PROGRAM MAIN
VAR
	bCoinEnter 	: BOOL;
	bManual		: BOOL;
	bAuto		: BOOL;
	bLedPower	: BOOL;

	bPlainWater	: BOOL:=TRUE;
	bLedW		: BOOL;
	
	bShampoo	: BOOL:=TRUE;
	bLedS		: BOOL;

    bWax		: BOOL:=TRUE;
	bLedWx		: BOOL;
	
	tRunningTimeM	: TIME:=T#9S;
	tTimer 		: TOF;	
	
	
END_VAR

IF bCoinEnter THEN
	
	//While process chosen as manual mode
	IF bManual THEN
		
		tTimer(IN:=bPlainWater AND bShampoo AND bWax,PT:= tRunningTimeM );
		//cCounter(CU:=tTimer.Q, RESET:= bCoinEnter, PV:=CounterPV );
		bLedPower		:= tTimer.Q;
	
		
		IF NOT bPlainWater THEN	  
		   bLedW		:= tTimer.Q;
    	   bShampoo		:= TRUE;
	   	   bWax			:= TRUE;
	 
       ELSIF NOT  bShampoo THEN	   
	   	  bLedS			:= tTimer.Q;  
	  	  bPlainWater	:= TRUE;
	      bWax			:= TRUE;
		  
   	  ELSIF NOT bWax THEN   	   
	      bLedWx		:= tTimer.Q;  
	      bShampoo		:= TRUE;
	      bPlainWater	:= TRUE;

      END_IF
  
      IF NOT tTimer.Q THEN
	    bCoinEnter 		:=FALSE;
	   	bPlainWater		:=TRUE;
		bShampoo		:=TRUE;
    	bWax			:=TRUE;
		bManual			:=FALSE;
		tTimer(IN:=TRUE);
		
		  
      END_IF
	   
	END_IF 
	
	
	
	
	//While process chosen as automatic mode
	IF bAuto THEN
		
		tTimer(IN:=FALSE,PT:= tRunningTimeM );
		bLedPower		:= tTimer.Q;
		
		IF tTimer.ET <= T#3S THEN
			bLedW			:= tTimer.Q;
			
        ELSIF tTimer.ET <= T#6S THEN
			bLedS			:= tTimer.Q;
			bLedW			:= FALSE;
 
			
		ELSIF tTimer.ET <= T#9S THEN
			bLedWx			:= tTimer.Q;
			bLedW			:= FALSE;
			bLedS			:= FALSE;
			
			
			
		END_IF
		
		
		IF NOT tTimer.Q THEN
	   	 	bCoinEnter 		:=FALSE;
			bLedW			:=FALSE;
			bLedS			:=FALSE;
            bLedWx			:=FALSE;
			bAuto			:=FALSE;
			tTimer(IN:=TRUE);
        END_IF
		
	END_IF
	
END_IF

END_PROGRAM

(* stored: Version 1.1.0.1, ProductVersion 3.1.4024.9
   POU MAIN: Id {fb19dc3b-8e79-4d2e-a250-880528b3d535}, SpecialFunc None *)
